Staubli VAL3: OnF3.pgx

program OnF3()
  local string l_sYesNo[2]
  local num l_i
begin

  //
  if sList[nSelected]!=""
    l_sYesNo[0]="是"
    l_sYesNo[1]="否"
    call user:questionDialog("是否删除?",l_sYesNo,l_i)
    if l_i==0 or l_i==1
      switch nPage
        case 0
          if size(sPrd)==1
            sPrd[nSelected]=""
            sProductList[nSelected]=""
          else
            delete(sPrd[nSelected])
            delete(sProductList[nSelected])
            if nSelected>=1
              nSelected=nSelected-1
            endIf
          endIf

        break
        case 1
          if size(sList)==1
            sList[nSelected]=""
          else
            delete(sList[nSelected])
            if nSelected>=1
              nSelected=nSelected-1
            endIf

          endIf
        break
      endSwitch
      bListRefresh=true
    else
      popUpMsg("没有可以删除的项目")
    endIf
  endIf
  bUserRefresh=true
end
